// TIA Portal V16 export
// export: Created 2022-09-29T14:55:01.2790762Z, ExportSetting WithDefaults, DisplayName Totally Integrated Automation Portal, DisplayVersion V16, DisplayName TIA Portal Version Control Interface, DisplayVersion V16, DisplayName TIA Portal Openness, DisplayVersion V16, DisplayName STEP 7 Professional, DisplayVersion V16, DisplayName STEP 7 Safety, DisplayVersion V16, DisplayName WinCC Advanced, DisplayVersion V16
DATA_BLOCK "Estados_HMI_DB"   // DB15
{ S7_Optimized_Access := 'TRUE' }
VERSION : 0.1
// stored: AutoNumber true, IsOnlyStoredInLoadMemory false, IsRetainMemResEnabled false, IsWriteProtectedInAS false, MemoryReserve 100
   VAR
      MX201 : Bool;
      MX601 : Bool;
      XV101 : Bool;
      XV102 : Bool;
      BD601 : Bool;
      BD602 : Bool;
      BH201 : Bool;
      PH201 : Bool;
      RH201 : Bool;
      MX603 : Bool;
      BD603 : Bool;
      MX301 : Bool;
      PH301 : Bool;
      BM401 : Bool;
      MX604 : Bool;
      BD604 : Bool;
      MX605 : Bool;
      BD605 : Bool;
      BS001A : Bool;
      BS001B : Bool;
      BS501 : Bool;
      T_ATUAL_AREJAMENTO : Time;
      T_ATUAL_REDUÇÃO : Time;
      T_ATUAL_PRECIPITAÇÃO : Time;
      T_ATUAL_ALARME_PC401 : Time;
      T_ATUAL_COAG : Time;
      T_ATUAL_HISTERESE : Time;
   END_VAR
BEGIN
END_DATA_BLOCK
